ABB RobotStudio station: Step_vacum_gripperV1.0.rspag

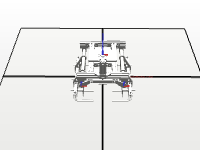
Station Step_suction_gripper (saved by RobotStudio 6.8.8307.1040)
Controller IRB_120_3kg_0.58m_1
  mechanical unit ROB_1: IRB120_3_58__01, 6 joints, base frame (0, 0, 0) mm
Layout (positions relative to the parent item):
  - IRB120_3_58__01 [mechanism] at (0, 0, 0) mm; joint values [0, 0, 0, 0, 0.5236, 0] (rad or m)
      links: Base, Link1, Link2, Link3, Link4, Link5, Link6
  - SmartComponent_1 [smart component]
    - toolgripper [mechanism] at (0, 0, 0) mm
        TCP L1 at (1038.22, -338, 221.07) mm
        TCP L2 at (652.5, -338, 219.93) mm
        TCP L3 at (845, -2.5, 337.43) mm
        links: T_GRIPPER v1
